DATA_BLOCK DB_TYPE_ADMIN
    STRUCT
        ProcessProfiles : ARRAY [1..10] OF UDT_PROCESS_PROFILE;
    END_STRUCT
BEGIN

END_DATA_BLOCK

